{attribute 'pack_mode' = '1'}
TYPE ST_AnyType :
STRUCT
	pValue : PVOID;
	nSize  : DINT;
END_STRUCT
END_TYPE

(* stored: Version 1.1.0.1, ProductVersion 3.1.4024.12
   DUT ST_AnyType: Id {2f218d5b-ad10-4c5f-9eba-9f839d114d28} *)
